// TIA Portal V16 export
// export: Created 2021-07-03T21:22:42.8322165Z, ExportSetting WithDefaults, DisplayName Totally Integrated Automation Portal, DisplayVersion V16, DisplayName TIA Portal Version Control Interface, DisplayVersion V16, DisplayName TIA Portal Openness, DisplayVersion V16, DisplayName STEP 7 Professional, DisplayVersion V16, DisplayName STEP 7 Safety, DisplayVersion V16, DisplayName WinCC Professional, DisplayVersion V16
TYPE "118MK2_RecipeData"
// stored: IsFailsafeCompliant false
   STRUCT
      REC1_EJEC_DELAY_TIME : Byte;   // Recipe-1: Ejector delay time - Unsigned 8 bit integer value. Range 0 to 50ms
      REC1_EJEC_ON_TIME : Byte;   // Recipe-1: Ejector on time - Unsigned 8 bit integer value. Range 1 to 50ms
      REC1_ALG_BLINT_TH : Word;   // Recipe-1: Algorithm blue intensity threshold - Unsigned 16 bit integer value. Range 60 to 10000mV
      REC1_ALG_BLRED_DISC_OFF : Word;   // Recipe-1: Algorithm blue-red discrimination offset - Unsigned 16 bit integer value. Range 0 to 10000
      REC1_ALG_BLRED_DISC_RAT : Word;   // Recipe-1: Algorithm blue-red discrimination ratio - Unsigned 16 bit integer value. Range 1 to 1000 (is gradient of 0.01 to 10.00)
      REC1_VIB_FEED_SP : Byte;   // Recipe-1: Vibratory feeder set-point, Unsigned 8 bit integer value. Range 0 to 100%
      REC1_AUTO_FEED_CNTRL : Bool;   // Recipe-1: Automatic feeder control - OFF(0) – No closed loop control, ON(1) – Closed loop control
      REC1_RESERVED1 : Bool;   // Recipe-1: Reserved - Spare
      REC1_RESERVED2 : Bool;   // Recipe-1: Reserved - Spare
      REC1_RESERVED3 : Bool;   // Recipe-1: Reserved - Spare
      REC1_RESERVED4 : Bool;   // Recipe-1: Reserved - Spare
      REC1_RESERVED5 : Bool;   // Recipe-1: Reserved - Spare
      REC1_RESERVED6 : Bool;   // Recipe-1: Reserved - Spare
      REC1_RESERVED7 : Bool;   // Recipe-1: Reserved - Spare
      REC1_GATE_POSITION : Byte;   // Recipe-1: Gate position - Range 0 to 5, ‘0’ - No auto gate control, ‘1’ – Move gate to position 1(-2 +1mm), ‘2’ – Move gate to position 2(-4+2mm), ‘3’ – Move gate to position 3(-8+4mm), ‘4’ – Move gate to position 4(-16+8mm), ‘5’ – Move gate to position 5(-32+16mm)
      SPARE0 : Byte;   // Spare
      SPARE1 : Word;   // Spare
      REC2_EJEC_DELAY_TIME : Byte;   // Recipe-2: Ejector delay time - Unsigned 8 bit integer value. Range 0 to 50ms
      REC2_EJEC_ON_TIME : Byte;   // Recipe-2: Ejector on time - Unsigned 8 bit integer value. Range 1 to 50ms
      REC2_ALG_BLINT_TH : Word;   // Recipe-2: Algorithm blue intensity threshold - Unsigned 16 bit integer value. Range 60 to 10000mV
      REC2_ALG_BLRED_DISC_OFF : Word;   // Recipe-2: Algorithm blue-red discrimination offset - Unsigned 16 bit integer value. Range 0 to 10000
      REC2_ALG_BLRED_DISC_RAT : Word;   // Recipe-2: Algorithm blue-red discrimination ratio - Unsigned 16 bit integer value. Range 1 to 1000 (is gradient of 0.01 to 10.00)
      REC2_VIB_FEED_SP : Byte;   // Recipe-2: Vibratory feeder set-point, Unsigned 8 bit integer value. Range 0 to 100%
      REC2_AUTO_FEED_CNTRL : Bool;   // Recipe-2: Automatic feeder control - OFF(0) – No closed loop control, ON(1) – Closed loop control
      REC2_RESERVED1 : Bool;   // Recipe-2: Reserved - Spare
      REC2_RESERVED2 : Bool;   // Recipe-2: Reserved - Spare
      REC2_RESERVED3 : Bool;   // Recipe-2: Reserved - Spare
      REC2_RESERVED4 : Bool;   // Recipe-2: Reserved - Spare
      REC2_RESERVED5 : Bool;   // Recipe-2: Reserved - Spare
      REC2_RESERVED6 : Bool;   // Recipe-2: Reserved - Spare
      REC2_RESERVED7 : Bool;   // Recipe-2: Reserved - Spare
      REC2_GATE_POSITION : Byte;   // Recipe-2: Gate position - Range 0 to 5, ‘0’ - No auto gate control, ‘1’ – Move gate to position 1(-2 +1mm), ‘2’ – Move gate to position 2(-4+2mm), ‘3’ – Move gate to position 3(-8+4mm), ‘4’ – Move gate to position 4(-16+8mm), ‘5’ – Move gate to position 5(-32+16mm)
      SPARE2 : Byte;   // Spare
      SPARE3 : Word;   // Spare
      REC3_EJEC_DELAY_TIME : Byte;   // Recipe-3: Ejector delay time - Unsigned 8 bit integer value. Range 0 to 50ms
      REC3_EJEC_ON_TIME : Byte;   // Recipe-3: Ejector on time - Unsigned 8 bit integer value. Range 1 to 50ms
      REC3_ALG_BLINT_TH : Word;   // Recipe-3: Algorithm blue intensity threshold - Unsigned 16 bit integer value. Range 60 to 10000mV
      REC3_ALG_BLRED_DISC_OFF : Word;   // Recipe-3: Algorithm blue-red discrimination offset - Unsigned 16 bit integer value. Range 0 to 10000
      REC3_ALG_BLRED_DISC_RAT : Word;   // Recipe-3: Algorithm blue-red discrimination ratio - Unsigned 16 bit integer value. Range 1 to 1000 (is gradient of 0.01 to 10.00)
      REC3_VIB_FEED_SP_1 : Byte;   // Recipe-3: Vibratory feeder set-point, Unsigned 8 bit integer value. Range 0 to 100%
      REC3_AUTO_FEED_CNTRL : Bool;   // Recipe-3: Automatic feeder control - OFF(0) – No closed loop control, ON(1) – Closed loop control
      REC3_RESERVED1 : Bool;   // Recipe-3: Reserved - Spare
      REC3_RESERVED2 : Bool;   // Recipe-3: Reserved - Spare
      REC3_RESERVED3 : Bool;   // Recipe-3: Reserved - Spare
      REC3_RESERVED4 : Bool;   // Recipe-3: Reserved - Spare
      REC3_RESERVED5 : Bool;   // Recipe-3: Reserved - Spare
      REC3_RESERVED6 : Bool;   // Recipe-3: Reserved - Spare
      REC3_RESERVED7 : Bool;   // Recipe-3: Reserved - Spare
      REC3_GATE_POSITION : Byte;   // Recipe-3: Gate position - Range 0 to 5, ‘0’ - No auto gate control, ‘1’ – Move gate to position 1(-2 +1mm), ‘2’ – Move gate to position 2(-4+2mm), ‘3’ – Move gate to position 3(-8+4mm), ‘4’ – Move gate to position 4(-16+8mm), ‘5’ – Move gate to position 5(-32+16mm)
      SPARE4 : Byte;   // Spare
      SPARE5 : Word;   // Spare
      REC4_EJEC_DELAY_TIME : Byte;   // Recipe-4: Ejector delay time - Unsigned 8 bit integer value. Range 0 to 50ms
      REC4_EJEC_ON_TIME : Byte;   // Recipe-4: Ejector on time - Unsigned 8 bit integer value. Range 1 to 50ms
      REC4_ALG_BLINT_TH : Word;   // Recipe-4: Algorithm blue intensity threshold - Unsigned 16 bit integer value. Range 60 to 10000mV
      REC4_ALG_BLRED_DISC_OFF : Word;   // Recipe-4: Algorithm blue-red discrimination offset - Unsigned 16 bit integer value. Range 0 to 10000
      REC4_ALG_BLRED_DISC_RAT : Word;   // Recipe-4: Algorithm blue-red discrimination ratio - Unsigned 16 bit integer value. Range 1 to 1000 (is gradient of 0.01 to 10.00)
      REC4_VIB_FEED_SP : Byte;   // Recipe-4: Vibratory feeder set-point, Unsigned 8 bit integer value. Range 0 to 100%
      REC4_AUTO_FEED_CNTRL : Bool;   // Recipe-4: Automatic feeder control - OFF(0) – No closed loop control, ON(1) – Closed loop control
      REC4_RESERVED1 : Bool;   // Recipe-4: Reserved - Spare
      REC4_RESERVED2 : Bool;   // Recipe-4: Reserved - Spare
      REC4_RESERVED3 : Bool;   // Recipe-4: Reserved - Spare
      REC4_RESERVED4 : Bool;   // Recipe-4: Reserved - Spare
      REC4_RESERVED5 : Bool;   // Recipe-4: Reserved - Spare
      REC4_RESERVED6 : Bool;   // Recipe-4: Reserved - Spare
      REC4_RESERVED7 : Bool;   // Recipe-4: Reserved - Spare
      REC4_GATE_POSITION : Byte;   // Recipe-4: Gate position - Range 0 to 5, ‘0’ - No auto gate control, ‘1’ – Move gate to position 1(-2 +1mm), ‘2’ – Move gate to position 2(-4+2mm), ‘3’ – Move gate to position 3(-8+4mm), ‘4’ – Move gate to position 4(-16+8mm), ‘5’ – Move gate to position 5(-32+16mm)
      SPARE6 : Byte;   // Spare
      SPARE7 : Word;   // Spare
      REC5_EJEC_DELAY_TIME : Byte;   // Recipe-5: Ejector delay time - Unsigned 8 bit integer value. Range 0 to 50ms
      REC5_EJEC_ON_TIME : Byte;   // Recipe-5: Ejector on time - Unsigned 8 bit integer value. Range 1 to 50ms
      REC5_ALG_BLINT_TH : Word;   // Recipe-5: Algorithm blue intensity threshold - Unsigned 16 bit integer value. Range 60 to 10000mV
      REC5_ALG_BLRED_DISC_OFF : Word;   // Recipe-5: Algorithm blue-red discrimination offset - Unsigned 16 bit integer value. Range 0 to 10000
      REC5_ALG_BLRED_DISC_RAT : Word;   // Recipe-5: Algorithm blue-red discrimination ratio - Unsigned 16 bit integer value. Range 1 to 1000 (is gradient of 0.01 to 10.00)
      REC5_VIB_FEED_SP : Byte;   // Recipe-5: Vibratory feeder set-point, Unsigned 8 bit integer value. Range 0 to 100%
      REC5_AUTO_FEED_CNTRL : Bool;   // Recipe-5: Automatic feeder control - OFF(0) – No closed loop control, ON(1) – Closed loop control
      REC5_RESERVED1 { ExternalAccessible := 'False'; ExternalVisible := 'False'; ExternalWritable := 'False'} : Bool;   // Recipe-5: Reserved - Spare
      REC5_RESERVED2 { ExternalAccessible := 'False'; ExternalVisible := 'False'; ExternalWritable := 'False'} : Bool;   // Recipe-5: Reserved - Spare
      REC5_RESERVED3 { ExternalAccessible := 'False'; ExternalVisible := 'False'; ExternalWritable := 'False'} : Bool;   // Recipe-5: Reserved - Spare
      REC5_RESERVED4 { ExternalAccessible := 'False'; ExternalVisible := 'False'; ExternalWritable := 'False'} : Bool;   // Recipe-5: Reserved - Spare
      REC5_RESERVED5 { ExternalAccessible := 'False'; ExternalVisible := 'False'; ExternalWritable := 'False'} : Bool;   // Recipe-5: Reserved - Spare
      REC5_RESERVED6 { ExternalAccessible := 'False'; ExternalVisible := 'False'; ExternalWritable := 'False'} : Bool;   // Recipe-5: Reserved - Spare
      REC5_RESERVED7 { ExternalAccessible := 'False'; ExternalVisible := 'False'; ExternalWritable := 'False'} : Bool;   // Recipe-5: Reserved - Spare
      REC5_GATE_POSITION { ExternalAccessible := 'False'; ExternalVisible := 'False'; ExternalWritable := 'False'} : Byte;   // Recipe-5: Gate position - Range 0 to 5, ‘0’ - No auto gate control, ‘1’ – Move gate to position 1(-2 +1mm), ‘2’ – Move gate to position 2(-4+2mm), ‘3’ – Move gate to position 3(-8+4mm), ‘4’ – Move gate to position 4(-16+8mm), ‘5’ – Move gate to position 5(-32+16mm)
      SPARE8 { ExternalAccessible := 'False'; ExternalVisible := 'False'; ExternalWritable := 'False'} : Byte;   // Spare
      SPARE9 { ExternalAccessible := 'False'; ExternalVisible := 'False'; ExternalWritable := 'False'} : Word;   // Spare
   END_STRUCT;
END_TYPE
